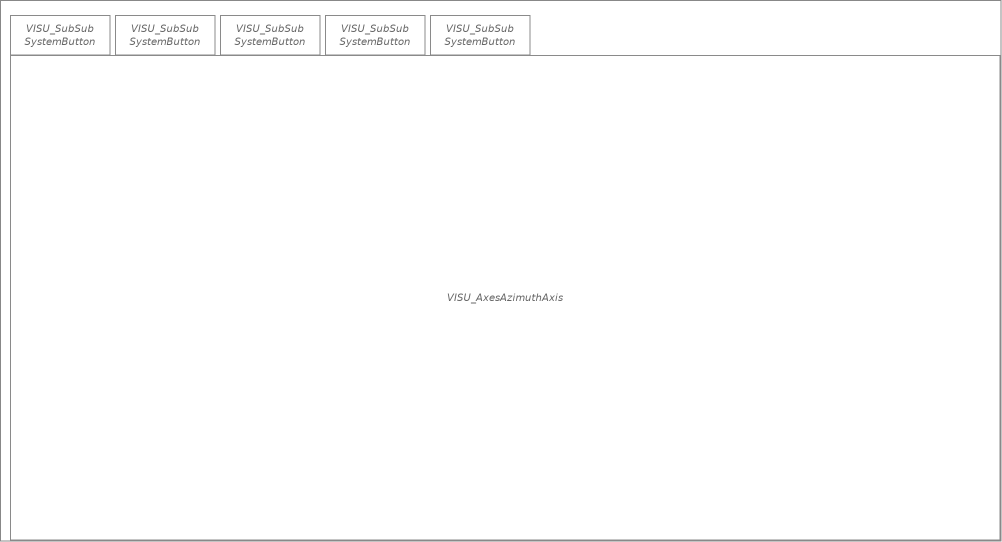
VISUALIZATION VISU_AxesAxes  // 1002x542
VAR_IN_OUT
    ref : Axes;
    widget : AxesAxesWidget;
END_VAR
    Frame (10,15 100x40)
        shows VISU_SubSubSystemButton(widget := widget.button_azi)
        OnMouseClick: FrameSelectionChange Selection=SelectedFrame=849b1b6c-774b-4476-bff7-38dbb17a175e, GlobSel=AssignType=Directly, SelType=Locally
        OnMouseClick: execute { widget.activeTab := AxesAxesTabs.AZI; }
    Frame (10,55 990x485)
        shows VISU_AxesAzimuthAxis(ref := ref.parts.azi, ref_aziDriveChannel := ref.parts.io.parts.aziDrive.parts.channelA, ref_ablDriveChannel := ref.parts.io.parts.ablDrive.parts.channelA, widget := widget.azi)
        shows VISU_AxesElevationAxis(ref := ref.parts.ele, ref_driveChannel := ref.parts.io.parts.eleDrive.parts.channelA, widget := widget.ele)
        shows VISU_AxesRotationAxis(ref := ref.parts.roc, ref_driveChannel := ref.parts.io.parts.aziDrive.parts.channelB, widget := widget.roc)
        shows VISU_AxesRotationAxis(ref := ref.parts.ron, ref_driveChannel := ref.parts.io.parts.ablDrive.parts.channelB, widget := widget.ron)
    Frame (115,15 100x40)
        shows VISU_SubSubSystemButton(widget := widget.button_ele)
        OnMouseClick: FrameSelectionChange Selection=SelectedFrame=849b1b6c-774b-4476-bff7-38dbb17a175e, Selection=1, GlobSel=AssignType=Directly, SelType=Locally
        OnMouseClick: execute { widget.activeTab := AxesAxesTabs.ELE; }
    Frame (220,15 100x40)
        shows VISU_SubSubSystemButton(widget := widget.button_roc)
        OnMouseClick: FrameSelectionChange Selection=SelectedFrame=849b1b6c-774b-4476-bff7-38dbb17a175e, Selection=2, GlobSel=AssignType=Directly, SelType=Locally
        OnMouseClick: execute { widget.activeTab := AxesAxesTabs.ROC; }
    Frame (325,15 100x40)
        shows VISU_SubSubSystemButton(widget := widget.button_ron)
        OnMouseClick: FrameSelectionChange Selection=SelectedFrame=849b1b6c-774b-4476-bff7-38dbb17a175e, Selection=3, GlobSel=AssignType=Directly, SelType=Locally
        OnMouseClick: execute { widget.activeTab := AxesAxesTabs.RON; }
    Frame (430,15 100x40)
        shows VISU_SubSubSystemButton(widget := widget.button_fw)
        OnMouseClick: FrameSelectionChange Selection=SelectedFrame=849b1b6c-774b-4476-bff7-38dbb17a175e, GlobSel=AssignType=Directly, SelType=Locally
        OnMouseClick: execute { widget.activeTab := AxesAxesTabs.FW; }
END_VISUALIZATION

(* stored: Version 1.1.0.1, ProductVersion 3.1.4019.2
   Visu VISU_AxesAxes: Id {9de19861-9485-4cd8-b254-1555f1432a0f} *)
